FUNCTION_BLOCK Test_AggregateResult_ErrorMsg EXTENDS T_UnitTestBase
VAR
	ResultAggregate : T_ResultAggregate;
	Execution1 : T_Execution;
	Execution2 : T_Execution;
	Execution3 : T_Execution;
END_VAR

{attribute 'analysis' := '-33'} // inhibit unused variable warning
METHOD RunTest
IF Retest THEN
    SUPER^.Init();
END_IF

IF TestCompleted THEN
    RETURN;
END_IF

F_Inc(CycleCount);
IF CycleCount > 1000 THEN
    Fail(Message := 'Timeout');
END_IF

ResultAggregate.Clear();

ResultAggregate.AddResult(Execution1);
ResultAggregate.AddResult(Execution2);
ResultAggregate.AddResult(Execution3);

Execution1.Start();
Execution1.SetBusy();
Execution1.SetDone();

Execution2.Start();
Execution2.SetBusy();
Execution2.SetDone();

AssertIsTrue(Condition := ResultAggregate.ErrorMsg = '',
             Message   := 'ResultAggregate.ErrorMsg is not blank');

Execution3.Start();
Execution3.SetBusy();
Execution3.SetError('Expected Error Message');

AssertIsTrue(Condition := ResultAggregate.ErrorMsg = 'Expected Error Message',
             Message   := 'ResultAggregate.ErrorMsg is incorrect');

TestCompleted := TRUE;
END_METHOD

END_FUNCTION_BLOCK

(* stored: Version 1.1.0.1, ProductVersion 3.1.4024.15
   POU Test_AggregateResult_ErrorMsg: Id {d530d38e-298d-4b11-aec7-52b51919ea3d}, SpecialFunc None
   Method RunTest: Id {2220bc6c-d318-41e4-8ea4-16c66d67b531} *)
